                            ELSIF (instHome.Error = TRUE OR instTimerTON.Q) THEN
                                // Errorhandling
                                statStatus                    := ERR_MC_HOME;
                                statErrorAutoCleared          := TRUE;
                                diagnostics                   := statDiagnostics;
                                diagnostics.subfunctionStatus := instHome.ErrorId;
                                statFBState                   := AXIS_STOP_ON_ERROR_SELECTION;
                                statBasicMotionState          := NO_SELECTION;

                            ELSE
                                ; // Command selected

                            END_IF;

                            statExeOfBasicMotion   := 16#0;
                            statExeOfBasicMotion.0 := instHome.Busy;
                            statExeOfBasicMotion.1 := instHome.Done;
                            statExeOfBasicMotion.2 := instHome.CommandAborted;
                            statExeOfBasicMotion.3 := instHome.Error;
                        {END_REGION}
                        HOMING_ON_FIXED_STOP:
                            // This case is additional feature (MC_MOVEVELOCITY and MC_HOME internal used)
                            {REGION "REFERENCE_TO_FIXED_STOP"}
                            CASE statExeOfBasicMotion OF
                                CMD_BUSY:
                                    // Firstcycle of command
                                    IF (statFirstCycleBasicMotion = TRUE) THEN
                                        // Check if homing on fixed stop is allowed  
                                        (*IF ( axis.Modulo.Enable = TRUE) THEN*)
                                        IF (tempFalse = TRUE) THEN
                                            // Modulo enabled - Errorhandling
                                            statStatus                    := ERR_MODULO_NOT_ALLOWED;
                                            statErrorAutoCleared          := TRUE;
                                            diagnostics.subfunctionStatus := 0;
                                            diagnostics.basicMotionState  := statBasicMotionState;
                                            // Set next state
                                            statFBState           := AXIS_STOP_ON_ERROR_SELECTION;
                                            statBasicMotionState  := NO_SELECTION;
                                            statActiveHomingState := STANDARD_HOMING;
                                            statHomingSubState    := HOMING_IDLE;

                                        ELSIF (configuration.homing.extendedModeTorqueLimit = 0) // Torqueliming 0 in configuration 
                                            THEN
                                            // Errorhandling -  Torquevalue 0 configured
                                            statStatus                    := ERR_INVALID_TORQUE_LIMIT;
                                            statErrorAutoCleared          := TRUE;
                                            diagnostics.subfunctionStatus := 0;
                                            diagnostics.basicMotionState  := statBasicMotionState;
                                            // Set next state
                                            statFBState           := AXIS_STOP_ON_ERROR_SELECTION;
                                            statBasicMotionState  := NO_SELECTION;
                                            statActiveHomingState := STANDARD_HOMING;
                                            statHomingSubState    := HOMING_IDLE;

                                            (*ELSIF ( axis.Homing.ReferencingVelocity = 0)*)
                                        ELSIF (configuration.homing.offsetPositionVelocity = 0)
                                            THEN
                                            // Errorhandling -  Velocity 0 configured
                                            statStatus                    := ERR_INVALID_VELOCITY;
                                            statErrorAutoCleared          := TRUE;
                                            diagnostics.subfunctionStatus := 0;
                                            diagnostics.basicMotionState  := statBasicMotionState;
                                            // Set next state
                                            statFBState           := AXIS_STOP_ON_ERROR_SELECTION;
                                            statBasicMotionState  := NO_SELECTION;
                                            statActiveHomingState := STANDARD_HOMING;
                                            statHomingSubState    := HOMING_IDLE;

                                        ELSE
                                            // Store dynamic values
                                            (*statHomingPosition :=  configuration.homing.position;
	                             statVelocity :=  axis.Homing.ReferencingVelocity;
	                             statAcceleration :=  axis.DynamicDefaults.Acceleration;
	                             statDeceleration :=  axis.DynamicDefaults.Deceleration;
	                             statJerk :=  axis.DynamicDefaults.Jerk;
	                             statTorqueLimit :=  configuration.homing.extendedModeTorqueLimit;*)
                                            statHomingPosition := configuration.homing.position;
                                            statVelocity       := configuration.homing.offsetPositionVelocity;
                                            statAcceleration   := configuration.homing.offsetPositionAcceleration;
                                            statDeceleration   := configuration.homing.offsetPositonDeceleration;
                                            statJerk           := configuration.homing.offsetPositionJerk;
                                            statTorqueLimit    := configuration.homing.extendedModeTorqueLimit;

                                            // Detecting operating sensor
                                            (*
								FOR  tempIndex := 1 TO 4 DO
	                              IF  axis.StatusSensor[ tempIndex].Control = TRUE
	                              THEN
	                                EXIT;
	                              END_IF;
	                            END_FOR;
	                            *)
                                            (*IF ( axis.Sensor[ tempIndex].ActiveHoming.Direction = 0) // Positve direction configured
	                            THEN*)
                                            // Positive direction
                                            statDirection := FORWARD_DIR;
                                            (* ELSE
	                              // Negative direction
	                               statDirection :=  BACKWARD_DIR;
	                            END_IF;
	                            *)
                                            (*statTorqueLimitingState :=  FIXED_STOP_DETECTION_ACTIVE;*)
                                            // Reset MC_Commands
                                            instHome(Axis := axis,
                                                     bCalibrationCam := homingSensor,
                                                     Execute := FALSE);

                                            instMoveVelocity(Axis := axis,
                                                             Execute := FALSE);

                                            instMoveAbsolute(Axis := axis,
                                                             Execute := FALSE);

                                            // Reset TON
                                            instTimerTON(IN := FALSE,
                                                         PT := configuration.homing.homeExecutionTimeLimit);

                                            // Determine the encoder type
                                            (* tempIndex := 1;
	                             tempIndex := UDINT_TO_INT( axis.OperativeSensor);
	                            IF ( axis.Sensor[ tempIndex].Type =  INCREMENTAL_ENCODER) THEN
	                               statHomingMode :=  DIRECT_HOMING; // Direct homing (absolute)
	                            ELSE
	                               statHomingMode :=  ABSOLUTE_ENCODER_ADJUSTMENT;
	                            END_IF;
								*)
                                            // Use always direct homing
                                            // statHomingMode :=  DIRECT_HOMING; // Direct homing (absolute)
                                            // Set next state
                                            (*statHomingSubState :=  HOMING_FIXED_STOP_DETECTION;*)
                                            statHomingSubState := HOMING_PROCESS;
                                        END_IF;
                                    END_IF;

                                    // Call OF subStateMachine
                                    REPEAT
                                        CASE statHomingSubState OF
                                            HOMING_IDLE:
                                                tempStateChangeActive := FALSE;
                                                ; // Do nothing, inserted no exectution of homing if error occurred in first cycle

                                            HOMING_FIXED_STOP_DETECTION:
                                                tempStateChangeActive := FALSE;

                                                // Start axis to detect fixed stop
                                                instMoveVelocity(Axis := axis,
                                                                 Execute := TRUE,
                                                                 Velocity := statVelocity,
                                                                 Acceleration := statAcceleration,
                                                                 Deceleration := statDeceleration,
                                                                 Jerk := statJerk,
                                                (*PositionControlled := TRUE,*)
                                                (*Direction :=  statDirection*) );

                                                // Read Statusword only when not already read out
                                                IF (tempStatusWord = 16#0)
                                                    THEN
                                                    (*tempStatusWord :=  axis.StatusWord;*)
                                                    tempStatusWord := axis.NcToPlc.StateDWord;
                                                END_IF;

                                                // Evaluate MC_Command
                                                IF (tempStatusWord.30 = TRUE) THEN // inClamping = TRUE
                                                    // Fixed stop detected --> start homing process
                                                    statHomingSubState    := HOMING_PROCESS;
                                                    tempStateChangeActive := TRUE;

                                                ELSIF (instMoveVelocity.Error = TRUE) THEN
                                                    // Errorhandling
                                                    statStatus                    := ERR_MC_MOVEVELOCITY;
                                                    statErrorAutoCleared          := TRUE;
                                                    diagnostics                   := statDiagnostics;
                                                    diagnostics.subfunctionStatus := instMoveVelocity.ErrorId;
                                                    // Set next state
                                                    statFBState           := AXIS_STOP_ON_ERROR_SELECTION;
                                                    statBasicMotionState  := NO_SELECTION;
                                                    statActiveHomingState := STANDARD_HOMING;
                                                    statExeOfBasicMotion  := CMD_ERROR;
                                                    statHomingSubState    := HOMING_IDLE;

                                                ELSIF (instMoveVelocity.CommandAborted = TRUE) THEN
                                                    // Set next state
                                                    statExeOfBasicMotion := CMD_ABORTED;
                                                    statHomingSubState   := HOMING_IDLE;

                                                ELSE
                                                    ; // Wait for detecting fixed stop
                                                END_IF;

                                            HOMING_PROCESS:
                                                tempStateChangeActive := FALSE;
                                                // Execute MC_HOME
                                                instHome(Axis := axis,
                                                         bCalibrationCam := homingSensor,
                                                         Execute := TRUE,
                                                         Position := statHomingPosition,
                                                (*Mode :=  statHomingMode*) );

                                                //Call TON
                                                instTimerTON(IN := TRUE,
                                                             PT := configuration.homing.homeExecutionTimeLimit);

                                                // Evaluate MC_Command
                                                IF (instHome.Done = TRUE) THEN
                                                    // MC_HOME finished - Set next state
                                                    statHomingSubState    := HOMING_POSITION;
                                                    tempStateChangeActive := TRUE;
                                                    instTimerTON.IN       := FALSE;

                                                ELSIF (instHome.Error = TRUE OR instTimerTON.Q) THEN
                                                    // Errorhandling
                                                    statStatus                    := ERR_MC_HOME;
                                                    statErrorAutoCleared          := TRUE;
                                                    diagnostics                   := statDiagnostics;
                                                    diagnostics.subfunctionStatus := instHome.ErrorId;
                                                    // Set next state
                                                    statFBState          := AXIS_STOP_ON_ERROR_SELECTION;
                                                    statExeOfBasicMotion := CMD_ERROR;
                                                    statHomingSubState   := HOMING_IDLE;

                                                ELSIF (instHome.CommandAborted = TRUE) THEN
                                                    // Set next state
                                                    statExeOfBasicMotion := CMD_ABORTED;
                                                    statHomingSubState   := HOMING_IDLE;
                                                ELSE
                                                    ; // Wait for finish homing process
                                                END_IF;

                                            HOMING_POSITION:
                                                tempStateChangeActive := FALSE;

                                                statHomingPosition := configuration.homing.offsetPosition;
                                                statVelocity       := configuration.homing.offsetPositionVelocity;
                                                statAcceleration   := configuration.homing.offsetPositionAcceleration;
                                                statDeceleration   := configuration.homing.offsetPositonDeceleration;
                                                statJerk           := configuration.homing.offsetPositionJerk;

                                                // Execute moving to homeposition
                                                instMoveAbsolute(Axis := axis,
                                                                 Execute := TRUE,
                                                                 (*Position :=  statHomingPosition,*)
                                                                 Position := configuration.homing.offsetPosition,
                                                                 Velocity := ABS(statVelocity),
                                                                 Acceleration := statAcceleration,
                                                                 Deceleration := statDeceleration,
                                                                 Jerk := statJerk,
                                                (*Direction :=  SHORTEST_WAY_DIR*) );

                                                // Evaluate MC_Command
                                                IF (instMoveAbsolute.Done = TRUE) THEN
                                                    // Homeposition reached - Set next state
                                                    statExeOfBasicMotion := CMD_DONE;
                                                    statHomingSubState   := HOMING_IDLE;

                                                ELSIF (instMoveAbsolute.Error = TRUE) THEN
                                                    // Errorhandling
                                                    statStatus                    := ERR_MC_MOVEABSOLUTE;
                                                    statErrorAutoCleared          := TRUE;
                                                    diagnostics                   := statDiagnostics;
                                                    diagnostics.subfunctionStatus := instMoveAbsolute.ErrorId;
                                                    // Set next state
                                                    statFBState           := AXIS_STOP_ON_ERROR_SELECTION;
                                                    statBasicMotionState  := CMD_BUSY;
                                                    statActiveHomingState := STANDARD_HOMING;
                                                    statExeOfBasicMotion  := CMD_ERROR;
                                                    statHomingSubState    := HOMING_IDLE;

                                                ELSIF (instMoveAbsolute.CommandAborted = TRUE) THEN
                                                    // Set next state
                                                    statExeOfBasicMotion := CMD_ABORTED;
                                                    statHomingSubState   := HOMING_IDLE;

                                                ELSE
                                                    ; // Wait for reaching homeposition
                                                END_IF;

                                        ELSE
                                            // Errorhandling 
                                            statStatus                    := ERR_UNDEFINED_EXTENDED_HOMING_SUBSTATE;
                                            statErrorUserCleared          := TRUE;
                                            diagnostics                   := statDiagnostics;
                                            diagnostics.subfunctionStatus := 0;
                                            // Set errorstate
                                            statFBState           := FB_ERROR;
                                            tempStateChangeActive := FALSE;
                                        END_CASE;

                                    UNTIL (tempStateChangeActive = FALSE) // Repeat execution if a state is changing
                                    END_REPEAT;

                                CMD_DONE,
                                    CMD_ABORTED,
                                    CMD_ERROR:
                                    // Return to NO_SELECTION if command finished
                                    IF (statBasicCommand.10 = FALSE) // homing = FALSE
                                        THEN
                                        // Return to NO_HOMING_ACTIVE if command finished
                                        statBasicMotionState  := NO_SELECTION;
                                        statActiveHomingState := STANDARD_HOMING;
                                        statExeOfBasicMotion  := CMD_BUSY;
                                        statHomingSubState    := HOMING_IDLE;
                                    ELSE
                                        ; // Wait for falling edge at homing command
                                    END_IF;

                            ELSE
                                // Errorhandling
                                statStatus                    := ERR_UNDEFINED_EXTENDED_HOMING_STATE;
                                statErrorUserCleared          := TRUE;
                                diagnostics                   := statDiagnostics;
                                diagnostics.subfunctionStatus := 0;
                                // Set errorstate
                                statFBState := FB_ERROR;
                            END_CASE;
                    {END_REGION}

                    ELSE
                        // Errorhandling
                        statStatus                    := ERR_INVALID_HOMING_EXTENDED_MODE;
                        statErrorAutoCleared          := TRUE;
                        diagnostics                   := statDiagnostics;
                        diagnostics.subfunctionStatus := 0;
                        // Set next state
                        statFBState           := AXIS_STOP_ON_ERROR_SELECTION;
                        statBasicMotionState  := NO_SELECTION;
                        statActiveHomingState := STANDARD_HOMING;
                        statBasicMotionState  := NO_SELECTION;
                    END_CASE;
                {END_REGION}

                GEAR_IN_RELATIVE_SELECTED:
                    // Additional features (applicative): Change setpoint on the fly (gear ratio)
                    {REGION "GEAR_IN_RELATIVE_SELECTED"}
                    // Firstcycle of command
                    IF (statFirstCycleBasicMotion = TRUE) THEN
                        // Reset GEAR_IN command 
                        instGearIn(Master := master,
                                   Slave := axis,
                                   Execute := FALSE);

                        (*statRatioNumerator :=  configuration.gearInRelative.ratioNumerator;*)
                        statRatioNumerator      := configuration.gearInRelative.ratioDenominator;
                        statRatioDenominator    := configuration.gearInRelative.ratioDenominator;
                        statAcceleration        := configuration.gearInRelative.acceleration;
                        statDeceleration        := configuration.gearInRelative.deceleration;
                        statJerk                := configuration.gearInRelative.jerk;
                        statRatioChangeOnTheFly := configuration.gearInRelative.ratioChangeOnTheFly;

                    ELSIF ((statRatioChangeOnTheFly = TRUE) // Flying change of ratio numerator
                    (*AND (( configuration.gearInRelative.ratioNumerator <>  statRatioNumerator)*)
                        AND
                        ((configuration.gearInRelative.ratioDenominator <> statRatioNumerator) OR
                        (configuration.gearInRelative.ratioDenominator <> statRatioDenominator))) AND
                        (instGearIn.CommandAborted = FALSE)
                        THEN
                        instGearIn(Master := master,
                                   Slave := axis,
                                   Execute := FALSE);

                        statRatioNumerator   := configuration.gearInRelative.ratioDenominator; // Apply the new gear ratio numerator
                        statRatioDenominator := configuration.gearInRelative.ratioDenominator; // Apply the new gear ratio denominator
                    END_IF;

                    // Call MC_Command
                    instGearIn(Master := master,
                               Slave := axis,
                               Execute := statBasicCommand.7 OR statFirstCycleBasicMotion, // Input: gearInRelative
                               RatioNumerator := statRatioNumerator,
                               RatioDenominator := DINT_TO_UINT(statRatioDenominator),
                               Acceleration := statAcceleration,
                               Deceleration := statDeceleration,
                               Jerk := statJerk);

                    // Evaluate MC_Command
                    IF (instGearIn.Busy = FALSE) AND
                        (instGearIn.Error = FALSE) AND
                        (instGearIn.CommandAborted = FALSE) AND
                        (instGearIn.InGear = FALSE)
                        THEN
                        // Return to NO_SELECTION if command finished
                        statBasicMotionState := NO_SELECTION;

                    ELSIF (instGearIn.Error = TRUE) THEN
                        // Errorhandling
                        statStatus                    := ERR_MC_GEARIN;
                        statErrorAutoCleared          := TRUE;
                        diagnostics                   := statDiagnostics;
                        diagnostics.subfunctionStatus := instGearIn.ErrorId;
                        statRatioChangeOnTheFly       := FALSE;
                        // Set next state
                        statFBState          := AXIS_STOP_ON_ERROR_SELECTION;
                        statBasicMotionState := NO_SELECTION;

                    ELSE
                        ; // Command selected
                    END_IF;

                    // Read Statusword only when not already read out
                    // IF ( tempStatusWord = 16#0)
                    // THEN
                    //    tempStatusWord :=  axis.StatusWord;
                    // END_IF;

                    // Write MC_Command outputs to internal variable
                    statExeOfBasicMotion   := 16#0;
                    statExeOfBasicMotion.0 := instGearIn.Busy;
                    statExeOfBasicMotion.2 := instGearIn.CommandAborted;
                    statExeOfBasicMotion.3 := instGearIn.Error;
                    // statExeOfBasicMotion.6 :=  tempStatusWord.21 AND NOT  instGearIn.InGear; // write Synchronizing only when bit of instance of MC_GearIn.InGear = FALSE
                    statExeOfBasicMotion.7 := instGearIn.InGear;
                {END_REGION}

                GEAR_IN_ABSOLUTE_SELECTED:
                    // Additional features (applicative): Change setpoint on the fly (gear ratio)
                    {REGION "GEAR_IN_SELECTED"}
                    // Firstcycle of command
                    IF (statFirstCycleBasicMotion = TRUE) THEN
                        // Reset GEAR_IN_POS command 
                        instGearInPos(Master := master,
                                      Slave := axis,
                        (*Execute := FALSE*) );

                        statRatioNumerator       := configuration.gearInAbsolute.ratioNumerator;
                        statRatioDenominator     := configuration.gearInAbsolute.ratioDenominator;
                        statMasterSyncPosition   := configuration.gearInAbsolute.masterSyncPosition;
                        statSlaveSyncPosition    := configuration.gearInAbsolute.slaveSyncPosition;
                        statSyncProfileReference := configuration.gearInAbsolute.syncProfileReference;
                        statMasterStartDistance  := configuration.gearInAbsolute.masterStartDistance;
                        statVelocity             := configuration.gearInAbsolute.velocity;
                        statAcceleration         := configuration.gearInAbsolute.acceleration;
                        statDeceleration         := configuration.gearInAbsolute.deceleration;
                        statJerk                 := configuration.gearInAbsolute.jerk;
                        statSyncDirection        := configuration.gearInAbsolute.syncDirection;
                        statRatioChangeOnTheFly  := configuration.gearInAbsolute.ratioChangeOnTheFly;

                    ELSIF (((statRatioChangeOnTheFly = TRUE) AND (configuration.gearInAbsolute.ratioNumerator <> statRatioNumerator)) OR
                        ((statRatioChangeOnTheFly = TRUE) AND (configuration.gearInAbsolute.ratioDenominator <> statRatioDenominator))) AND
                        (instGearInPos.CommandAborted = FALSE)
                        THEN
                        instGearInPos(Master := master,
                                      Slave := axis,
                        (*Execute := FALSE*) );

                        statRatioNumerator   := configuration.gearInAbsolute.ratioNumerator;   // Apply the new gear ratio numerator
                        statRatioDenominator := configuration.gearInAbsolute.ratioDenominator; // Apply the new gear ratio denominator
                    END_IF;

                    // Call MC_Command
                    instGearInPos(Master := master,
                                  Slave := axis,
                                  Enable := statBasicCommand.8 OR statFirstCycleBasicMotion, // Input: gearInAbsolute
                                  GearRatio := statRatioNumerator,
                                  (*RatioDenominator :=  statRatioDenominator,*)
                                  (*MasterSyncPosition :=  statMasterSyncPosition,*)
                                  (*SlaveSyncPosition :=  statSlaveSyncPosition,*)
                                  (*SyncProfileReference :=  statSyncProfileReference,*)
                                  (*MasterStartDistance :=  statMasterStartDistance,*)
                                  (*Velocity :=  statVelocity,*)
                                  (*Acceleration :=  statAcceleration,*)
                                  (*Deceleration :=  statDeceleration,*)
                                  Jerk := statJerk,
                    (*SyncDirection :=  statSyncDirection*) );

                    // Evaluate MC_Command
                    IF (instGearInPos.Busy = FALSE) AND
                        (instGearInPos.Error = FALSE) AND
                        (instGearInPos.CommandAborted = FALSE) AND
                    (*( instGearInPos.StartSync = FALSE) AND*)
                        (instGearInPos.InGear = FALSE)
                        THEN
                        // Return to NO_SELECTION if command finished
                        statBasicMotionState := NO_SELECTION;

                    ELSIF (instGearInPos.Error = TRUE) THEN
                        // Errorhandling
                        statStatus                    := ERR_MC_GEARINPOS;
                        statErrorAutoCleared          := TRUE;
                        diagnostics                   := statDiagnostics;
                        diagnostics.subfunctionStatus := instGearInPos.ErrorId;
                        statRatioChangeOnTheFly       := FALSE;
                        // Set next state
                        statFBState          := AXIS_STOP_ON_ERROR_SELECTION;
                        statBasicMotionState := NO_SELECTION;

                    ELSE
                        ; // Command selected
                    END_IF;

                    // Write MC_Command outputs to internal variable
                    statExeOfBasicMotion   := 16#0;
                    statExeOfBasicMotion.0 := instGearInPos.Busy;
                    statExeOfBasicMotion.2 := instGearInPos.CommandAborted;
                    statExeOfBasicMotion.3 := instGearInPos.Error;
                    (*statExeOfBasicMotion.6 :=  instGearInPos.StartSync;*)
                    (*statExeOfBasicMotion.6 :=  instGearInPos.StartSync;*)
                    statExeOfBasicMotion.7 := instGearInPos.InGear;
                {END_REGION}

                CAM_IN_SELECTED:
                    // Additional feature (applicative): Check DB of Cam 
                    {REGION "CAM_IN_SELECTED"}
                    // Firstcycle of command
                    IF (statFirstCycleBasicMotion = TRUE) THEN
                        (*IF TypeOfDB( cam) = TO_Cam*)
                        IF tempFalse = FALSE
                            THEN
                            (*statCam :=  cam;*)
                            // Reset CAM_IN command 
                            instCamIn(Master := master,
                                      Slave := axis,
                                      (*Cam :=  statCam,*)
                                      Execute := FALSE);

                            statApplicativeBasicMotionError := FALSE;
                            statApplicationMode             := configuration.camIn.applicationMode;
                        ELSE
                            // Errorhandling - Invalid cam
                            statStatus                      := ERR_INVALID_CAM;
                            statErrorAutoCleared            := TRUE;
                            diagnostics.subfunctionStatus   := 0;
                            diagnostics                     := statDiagnostics;
                            statApplicativeBasicMotionError := TRUE;
                            // Set next state
                            statFBState          := AXIS_STOP_ON_ERROR_SELECTION;
                            statBasicMotionState := NO_SELECTION;
                        END_IF;
                    END_IF;

                    IF (statApplicativeBasicMotionError = FALSE) THEN

                        // Write MC Parameters
                        instCamIn.CamTableID                 := configuration.camIn.tableID;
                        instCamIn.StartMode                  := configuration.camIn.startMode;
                        instCamIn.MasterOffset               := configuration.camIn.masterOffset;
                        instCamIn.SlaveOffset                := configuration.camIn.slaveOffset;
                        instCamIn.MasterScaling              := configuration.camIn.masterScaling;
                        instCamIn.SlaveScaling               := configuration.camIn.slaveScaling;
						instCamIn.StartMode     			 := configuration.camIn.startMode;
                        instCamIn.Options.ActivationMode     := configuration.camIn.ActivationMode;
                        instCamIn.Options.ActivationPosition := configuration.camIn.ActivationPosition;

                        // Call MC_Command
                        instCamIn(Master := master,
                                  Slave := axis,
                                  Execute := statBasicCommand.9 OR statFirstCycleBasicMotion);

                        // Evaluate MC_Command
                        IF ((instCamIn.Busy = FALSE) AND
                            (instCamIn.Error = FALSE) AND
                            (instCamIn.CommandAborted = FALSE) AND
                            (instCamIn.InSync = FALSE) AND
                        (*( instCamIn.StartSync = FALSE) AND*)
                            (statBasicCommand.9 = FALSE)
                            ) AND // V1.0.2 Wait for one cycle EndOfProfile (--> Done) before function is finished at applicationMode ONCE
                            ((statApplicationMode <> APPLICATION_MODE_ONCE) OR
                            ((statApplicationMode = APPLICATION_MODE_ONCE) (*AND ( instCamIn.EndOfProfile = FALSE)*) ))
                            THEN
                            // Return to NO_SELECTION if command finished
                            statBasicMotionState := NO_SELECTION;

                        ELSIF (instCamIn.Error = TRUE) THEN
                            // Errorhandling
                            statStatus                    := ERR_MC_CAMIN;
                            statErrorAutoCleared          := TRUE;
                            diagnostics.subfunctionStatus := instCamIn.ErrorId;
                            diagnostics.basicMotionState  := statBasicMotionState;
                            statFBState                   := AXIS_STOP_ON_ERROR_SELECTION;
                            statBasicMotionState          := NO_SELECTION;

                        ELSE
                            ; // Command selected
                        END_IF;

                        // Write MC_Command outputs to internal variable
                        statExeOfBasicMotion   := 16#0;
                        statExeOfBasicMotion.0 := instCamIn.Busy;
                        IF (statApplicationMode = APPLICATION_MODE_ONCE)
                            THEN
                            ; (*statExeOfBasicMotion.1 :=  instCamIn.EndOfProfile;*)
                        END_IF;

                        statExeOfBasicMotion.2 := instCamIn.CommandAborted;
                        statExeOfBasicMotion.3 := instCamIn.Error;
                        statExeOfBasicMotion.6 := NOT instCamIn.Active;
                        statExeOfBasicMotion.7 := instCamIn.InSync;

                    ELSE
                        ; // InValid cam
                    END_IF;
            {END_REGION}

            ELSE
                // Errorhandling
                statStatus                    := ERR_UNDEFINED_BASIC_MOTION_STATE;
                statErrorUserCleared          := TRUE;
                diagnostics                   := statDiagnostics;
                diagnostics.subfunctionStatus := 0;
                // Set errorstate
                statFBState := FB_ERROR;
            END_CASE;

        RESET_GEARING:
            // Abort waiting absolute gearing / camIn job if new basic motion job is selected (configuration.generalSettings.abortWaitingSyncCmd = TRUE)
            instGearIn(Master := master,
                       Slave := axis,
                       Execute := TRUE,
                       RatioNumerator := 1,
                       RatioDenominator := 1); // Lowest possible gear ratio

            IF (instGearIn.InGear = TRUE) OR (instGearIn.CommandAborted = TRUE)
                THEN                                            // Relative gearing command has aborted waiting absolute gearing job
                statMainSelectionState    := CALL_BASIC_MOTION; // Execute new basic motion command
                tempStateChangeActive     := TRUE;
                statFirstCycleBasicMotion := TRUE;

            ELSIF (instGearIn.Error = TRUE)
                THEN
                statStatus                    := ERR_MC_GEARIN;
                diagnostics.subfunctionStatus := instGearIn.ErrorId;
                // Errorhandling
                statErrorAutoCleared := TRUE;
                diagnostics          := statDiagnostics;
                // Set next state
                statFBState            := AXIS_STOP_ON_ERROR_SELECTION;
                statMainSelectionState := CALL_BASIC_MOTION;
                statBasicMotionState   := NO_SELECTION;

            ELSE
                ; // Command running
            END_IF;

            // Write MC_Command outputs to internal variable
            statExeOfBasicMotion   := 16#0;
            statExeOfBasicMotion.0 := instGearIn.Busy;
    ELSE
        // Errorhandling
        statStatus                    := ERR_UNDEFINED_MAIN_SELECTION_STATE;
        statErrorUserCleared          := TRUE;
        diagnostics                   := statDiagnostics;
        diagnostics.subfunctionStatus := 0;
        // Set errorstate
        statFBState := FB_ERROR;
    END_CASE;

UNTIL (tempStateChangeActive = FALSE)
END_REPEAT;

{END_REGION}

//----------------------------------------------------------------------------------------------
// Execution of homing functionality 
//----------------------------------------------------------------------------------------------
{REGION "EXECUTION_OF_PASSIVE_HOMING"}
// Statemachine for homing functionality
CASE statPassiveHomingState OF
    // Selection of extended homing mode  
    NO_HOMING_ACTIVE:
        ; // Do nothing

    STANDARD_HOMING:
        // No additional features
        {REGION "STANDARD_HOMING"}
        // Firstcycle of command
        IF (statFirstCycleHoming = TRUE) THEN
            // Reset MC_HOME command
            instHome(Axis := axis,
                     bCalibrationCam := homingSensor,
                     Execute := FALSE);

            IF (statBasicMotionState = ACTIVE_HOMING_SELECTED) THEN
                statBasicMotionState := NO_SELECTION;
            END_IF;
        END_IF;

        // Call MC_Command
        instHome(Axis := axis,
                 bCalibrationCam := homingSensor,
                 Execute := statExtendedCommand.2, // Input: homing
                 Position := configuration.homing.position,
        (*Mode :=  configuration.homing.mode*) );

        // Evaluate MC_Command
        IF (instHome.Busy = FALSE) AND
            (instHome.Done = FALSE) AND
            (instHome.CommandAborted = FALSE) AND
            (instHome.Error = FALSE)
            THEN
            // Return to NO_SELECTION if command finished
            statPassiveHomingState := NO_HOMING_ACTIVE;

        ELSIF (instHome.Error = TRUE) THEN
            // Errorhandling
            statStatus                    := ERR_MC_HOME;
            statErrorAutoCleared          := TRUE;
            diagnostics                   := statDiagnostics;
            diagnostics.subfunctionStatus := instHome.ErrorId;
            statPassiveHomingState        := NO_HOMING_ACTIVE;
            // Set next state
            statFBState := AXIS_STOP_ON_ERROR_SELECTION;
        ELSE
            ; // Command selected

        END_IF;

        statExeOfHoming   := 16#0;
        statExeOfHoming.0 := instHome.Busy;
        statExeOfHoming.1 := instHome.Done;
        statExeOfHoming.2 := instHome.CommandAborted;
        statExeOfHoming.3 := instHome.Error;
{END_REGION}

ELSE
    // Errorhandling
    statStatus                              := ERR_INVALID_HOMING_EXTENDED_MODE;
    statErrorAutoCleared                    := TRUE;
    diagnostics                             := statDiagnostics;
    diagnostics.subfunctionStatus           := 0;
    statDiagnostics.basicMotionState        := statBasicMotionState;
    statDiagnostics.superimposedMotionState := statSupImpMotionState;
    // Set next state
    statFBState            := AXIS_STOP_ON_ERROR_SELECTION;
    statBasicMotionState   := NO_SELECTION;
    statPassiveHomingState := NO_HOMING_ACTIVE;
END_CASE;

{END_REGION}

//----------------------------------------------------------------------------------------------
// Execution of functionalities of superimposed coordinate system
//----------------------------------------------------------------------------------------------
{REGION "EXECUTION_OF_SUPERIMPOSED_COMMANDS"}
// Statemachine for superimposed motion commands
// Write diagnostics
statDiagnostics.basicMotionState        := statBasicMotionState;
statDiagnostics.superimposedMotionState := statSupImpMotionState;

CASE statSupImpMotionState OF
    NO_SELECTION:
        ; // Do nothing

    POS_SUPERIMPOSED_SELECTED:
        // Additional features (applicative) : Specified direction
        {REGION "POS_SUPERIMPOSED_SELECTED;"}
        // Firstcycle of command
        IF (statFirstCycleSupImpMotion = TRUE) THEN
            // Configurate the direction of rotation
            IF ((configuration.posSuperimposed.direction = 0) AND (configuration.posSuperimposed.distance >= 0.0)) // Sign of distance is evaluated
                OR
                (configuration.posSuperimposed.direction = FORWARD_DIR) // Positive direction
                THEN
                statSupImpMotionPosition := ABS(configuration.posSuperimposed.distance);
                // Reset MC_MOVESUPERIMPOSED command
                instMoveSuperimposed(Axis := axis,
                                     Execute := FALSE);

                statApplicativeSupImpMotionError := FALSE;
            ELSIF ((configuration.posSuperimposed.direction = 0) AND (configuration.posSuperimposed.distance < 0.0)) // Sign of distance is evaluated
                OR
                (configuration.posSuperimposed.direction = BACKWARD_DIR) // Negative direction 
                THEN
                statSupImpMotionPosition := -ABS(configuration.posSuperimposed.distance);
                // Reset MC_MOVESUPERIMPOSED command
                instMoveSuperimposed(Axis := axis,
                                     Execute := FALSE);

                statApplicativeSupImpMotionError := FALSE;

            ELSE
                // Errorhandling - Invalid direction
                statStatus                       := ERR_INVALID_POS_SUPERIMPOSED_DIR;
                statErrorAutoCleared             := TRUE;
                diagnostics                      := statDiagnostics;
                diagnostics.subfunctionStatus    := 0;
                statApplicativeSupImpMotionError := TRUE;
                // Set next state
                statFBState           := AXIS_STOP_ON_ERROR_SELECTION;
                statSupImpMotionState := NO_SELECTION;
            END_IF;
        END_IF;

        IF (statApplicativeSupImpMotionError = FALSE) THEN
            // Call MC_Command
            instMoveSuperimposed(Axis := axis,
                                 Execute := statSupImpCommand.0, // Input: posSuperimposed
                                 Distance := statSupImpMotionPosition,
                                 VelocityDiff := configuration.posSuperimposed.velocityDiff,
                                 Acceleration := configuration.posSuperimposed.acceleration,
                                 Deceleration := configuration.posSuperimposed.deceleration,
                                 Jerk := configuration.posSuperimposed.jerk);

            // Evaluate MC_Command
            IF (instMoveSuperimposed.Busy = FALSE) AND
                (instMoveSuperimposed.Error = FALSE) AND
                (instMoveSuperimposed.Done = FALSE) AND
                (instMoveSuperimposed.CommandAborted = FALSE)
                THEN
                // Return to NO_SELECTION if command finished
                statSupImpMotionState := NO_SELECTION;

            ELSIF (instMoveSuperimposed.Error = TRUE) THEN
                // Errorhandling
                statStatus                    := ERR_MC_MOVESUPERIMPOSED;
                statErrorAutoCleared          := TRUE;
                diagnostics                   := statDiagnostics;
                diagnostics.subfunctionStatus := instMoveSuperimposed.ErrorId;
                // Set next state
                statFBState           := AXIS_STOP_ON_ERROR_SELECTION;
                statSupImpMotionState := NO_SELECTION;

            ELSE
                ; // command selected
            END_IF;

            statExeOfSupImpMotionState   := 16#0;
            statExeOfSupImpMotionState.0 := instMoveSuperimposed.Busy;
            statExeOfSupImpMotionState.1 := instMoveSuperimposed.Done;
            statExeOfSupImpMotionState.2 := instMoveSuperimposed.CommandAborted;
            statExeOfSupImpMotionState.3 := instMoveSuperimposed.Error;
        END_IF;
    {END_REGION}

    PHASING_SELECTED:
        // Additional features (applicative) : Change setpoint on the fly (phaseShift)
        {REGION "PHASING_SELECTED"}
        // Firstcycle of command
        IF (statFirstCycleSupImpMotion = TRUE) THEN
            // Reset MC_PHASING_ABSOLUTE command
            instPhasingAbsolute(Master := master,
                                Slave := axis,
                                Execute := FALSE);

            // Reset MC_PHASING_RELATIVE command
            instPhasingRelative(Master := master,
                                Slave := axis,
                                Execute := FALSE);

            statPhaseShift               := configuration.phasing.phaseShift;
            statVelocity                 := configuration.phasing.velocity;
            statAcceleration             := configuration.phasing.acceleration;
            statDeceleration             := configuration.phasing.deceleration;
            statJerk                     := configuration.phasing.jerk;
            statPhaseAbsolute            := configuration.phasing.phaseAbsolute;
            statChangePhaseShiftOnTheFly := configuration.phasing.phaseShiftChangeOnTheFly;

        ELSIF ((statChangePhaseShiftOnTheFly = TRUE) AND
            (configuration.phasing.phaseShift <> statPhaseShift)) AND
            (statPhaseAbsolute = TRUE) AND
            (instPhasingAbsolute.CommandAborted = FALSE)
            THEN
            // Reset MC_PHASING_ABSOLUTE command - Phaseshift on the fly is only possible at phasing absolut
            instPhasingAbsolute(Master := master,
                                Slave := axis,
                                Execute := FALSE);

            statPhaseShift := configuration.phasing.phaseShift;
        END_IF;

        // Select phasing absolut or relative 
        IF (statPhaseAbsolute = TRUE) THEN
            // Absolute phasing
            // Call MC_Command
            instPhasingAbsolute(Master := master,
                                Slave := axis,
                                Execute := statSupImpCommand.1, // Input: phasing
                                PhaseShift := statPhaseShift,
                                Velocity := statVelocity,
                                Acceleration := statAcceleration,
                                Deceleration := statDeceleration,
                                Jerk := statJerk);

            // Evaluate MC_Command
            IF (instPhasingAbsolute.Busy = FALSE) AND
                (instPhasingAbsolute.Error = FALSE) AND
                (instPhasingAbsolute.Done = FALSE) AND
                (instPhasingAbsolute.CommandAborted = FALSE)
                THEN
                // Return to NO_SELECTION if command finished
                statSupImpMotionState := NO_SELECTION;

            ELSIF (instPhasingAbsolute.Error = TRUE) THEN
                // Errorhandling
                statStatus                    := ERR_MC_PHASINGABSOLUTE;
                statErrorAutoCleared          := TRUE;
                diagnostics                   := statDiagnostics;
                diagnostics.subfunctionStatus := instPhasingAbsolute.ErrorId;
                statChangePhaseShiftOnTheFly  := FALSE;
                // Set next state
                statFBState           := AXIS_STOP_ON_ERROR_SELECTION;
                statSupImpMotionState := NO_SELECTION;

            ELSE
                ; // Command busy
            END_IF;

            statExeOfSupImpMotionState   := 16#0;
            statExeOfSupImpMotionState.0 := instPhasingAbsolute.Busy;
            statExeOfSupImpMotionState.1 := instPhasingAbsolute.Done;
            statExeOfSupImpMotionState.2 := instPhasingAbsolute.CommandAborted;
            statExeOfSupImpMotionState.3 := instPhasingAbsolute.Error;

        ELSE
            // Relative phasing  
            // Call MC_Command
            instPhasingRelative(Master := master,
                                Slave := axis,
                                Execute := statSupImpCommand.1, // Input: phasing
                                PhaseShift := statPhaseShift,
                                Velocity := statVelocity,
                                Acceleration := statAcceleration,
                                Deceleration := statDeceleration,
                                Jerk := statJerk);

            // Evaluate MC_Command
            IF (instPhasingRelative.Busy = FALSE) AND
                (instPhasingRelative.Error = FALSE) AND
                (instPhasingRelative.Done = FALSE) AND
                (instPhasingRelative.CommandAborted = FALSE)
                THEN
                // Return to NO_SELECTION if command finished
                statSupImpMotionState := NO_SELECTION;

            ELSIF (instPhasingRelative.Error = TRUE) THEN
                // Errorhandling
                statStatus                    := ERR_MC_PHASINGRELATIVE;
                statErrorAutoCleared          := TRUE;
                diagnostics                   := statDiagnostics;
                diagnostics.subfunctionStatus := instPhasingRelative.ErrorId;
                statChangePhaseShiftOnTheFly  := FALSE;
                // Set next state
                statFBState           := AXIS_STOP_ON_ERROR_SELECTION;
                statSupImpMotionState := NO_SELECTION;
            ELSE
                ; // Command selected
            END_IF;

            statExeOfSupImpMotionState   := 16#0;
            statExeOfSupImpMotionState.0 := instPhasingRelative.Busy;
            statExeOfSupImpMotionState.1 := instPhasingRelative.Done;
            statExeOfSupImpMotionState.2 := instPhasingRelative.CommandAborted;
            statExeOfSupImpMotionState.3 := instPhasingRelative.Error;
        END_IF;
{END_REGION}

ELSE
    // Errorhandling
    statStatus                    := ERR_UNDEFINED_SUPERIMPOSED_MOTION_STATE;
    statErrorUserCleared          := TRUE;
    diagnostics                   := statDiagnostics;
    diagnostics.subfunctionStatus := 0;
    // Set errorstate
    statFBState := FB_ERROR;
END_CASE;

{END_REGION}

//----------------------------------------------------------------------------------------------
// Execution of torquelimiting functionality
//----------------------------------------------------------------------------------------------
{REGION "EXECUTION_OF_TORQUELIMTING"}
// Statemachine for torquelimiting 
REPEAT
    tempStateChangeActive := FALSE;
    CASE statTorqueLimitingState OF
        NO_TORQUE_LIMITING_ACTIVE:
            ; // Torquelimiting disable
        //  instTorqueLimiting(Axis :=  axis, V01.00.03 Dont Call MC_TORQUELIMITING if disabled
        //                     Enable := FALSE);

        TORQUE_LIMITING_DISABLE:
            // Torquelimiting disable
            instTorqueLimiting(Axis := axis,
                               Enable := FALSE);

            // Check state of torque limting
            IF (instTorqueLimiting.Busy = FALSE)
                THEN
                // set next state
                statTorqueLimitingState := NO_TORQUE_LIMITING_ACTIVE;
            ELSE
                ; // Waiting for MC_Torquelimiting is not busy
            END_IF;

        TORQUE_LIMTING_SELECTED:
            // No extended homing function active
            instTorqueLimiting(Axis := axis,
                               Enable := statExtendedCommand.1,
                               TLimit := configuration.torqueLimiting.TorqueLimit,
                               Mode := configuration.torqueLimiting.mode);

            IF (instTorqueLimiting.Busy = FALSE) THEN
                // Reset state
                statTorqueLimitingState := NO_TORQUE_LIMITING_ACTIVE;
            END_IF;

        (*
	        V1.00.03 Not required anymore
	       AUTOMATIC_MODE_CHANGE:
	        // In this state the torquelimiting function is operating with Mode 1 (Fixed stop detection) until inClamping = FALSE
	         instTorqueLimiting(Axis :=  axis,
	                            Enable := TRUE,
	                            Limit :=  configuration.homing.extendedModeTorqueLimit); // V01.00.03 Always use configured value
	        
	        IF ( configuration.torqueLimiting.mode =  MODE_FIXED_STOP_DETECTION)
	          OR ( instTorqueLimiting.InClamping = FALSE)
	        THEN
	          // Change state
	           statTorqueLimitingState :=  TORQUE_LIMTING_SELECTED;
	           tempStateChangeActive := TRUE;
	        ELSE
	          ; // Wait for InClamping = FALSE
	        END_IF;
	        *)

        FIXED_STOP_DETECTION_ACTIVE:
            // Extended homing function active
            instTorqueLimiting(Axis := axis,
                               Enable := TRUE,
                               TLimit := configuration.homing.extendedModeTorqueLimit, // V01.00.03 Always use configured value
                               Mode := MODE_FIXED_STOP_DETECTION);

            IF ((statHomingSubState = HOMING_IDLE) AND (statBasicMotionState = ACTIVE_HOMING_SELECTED))
                THEN
                // Fixed stop process has finished - Axis is still in clamping
                statTorqueLimitingState := FIXED_STOP_DETECTION_FINISHED;
                tempStateChangeActive   := TRUE;

            ELSIF (statBasicMotionState <> ACTIVE_HOMING_SELECTED)
                THEN
                // Error occurred - change state depending on inClamping
                IF (instTorqueLimiting.InClamping = TRUE)
                    THEN
                    // Axis is in clamping
                    statTorqueLimitingState := FIXED_STOP_DETECTION_ERROR_IN_CLAMPING;
                    tempStateChangeActive   := TRUE;
                ELSE
                    // Axis is in not clamping
                    statTorqueLimitingState := FIXED_STOP_DETECTION_ERROR_NOT_IN_CLAMPING;
                    tempStateChangeActive   := TRUE;
                END_IF;

            ELSE
                ; // Fixed stop detection is running
            END_IF;

        FIXED_STOP_DETECTION_FINISHED:
            // Homing on fixed stop process has finished
            instTorqueLimiting(Axis := axis,
                               Enable := TRUE,
                               TLimit := configuration.homing.extendedModeTorqueLimit, // V01.00.03 Always use configured value
                               Mode := MODE_FIXED_STOP_DETECTION);

            IF (instTorqueLimiting.InClamping = FALSE)
                THEN
                // InClamping = FALSE
                IF (statExtendedCommand.1 = TRUE) // Torquelimiting
                    THEN
                    statTorqueLimitingState := TORQUE_LIMTING_SELECTED;
                ELSE
                    statTorqueLimitingState := TORQUE_LIMITING_DISABLE;
                END_IF;

                tempStateChangeActive := TRUE;
            ELSE
                // InClamping = TRUE
                IF (statExtendedCommand.1 = TRUE) // Torquelimiting
                    AND
                    (configuration.torqueLimiting.mode = MODE_FIXED_STOP_DETECTION)
                    THEN
                    // Change State
                    statTorqueLimitingState := TORQUE_LIMTING_SELECTED;
                    tempStateChangeActive   := TRUE;
                ELSE
                    ; // Wait for inClamping = FALSE
                END_IF;
            END_IF;

        FIXED_STOP_DETECTION_ERROR_IN_CLAMPING:
            // Errorstate, torquelimiting is still active and axis not in clamping
            instTorqueLimiting(Axis := axis,
                               Enable := TRUE,
                               TLimit := configuration.homing.extendedModeTorqueLimit, // V01.00.03 Always use configured value
                               Mode := MODE_FIXED_STOP_DETECTION);

            IF (instTorqueLimiting.InClamping = FALSE)
                THEN
                // InClamping = FALSE -> reset torque limiting state
                statTorqueLimitingState := TORQUE_LIMITING_DISABLE;
                // Torquelimiting disable
                tempStateChangeActive := TRUE;
            END_IF;

        FIXED_STOP_DETECTION_ERROR_NOT_IN_CLAMPING:
            // Errorstate, torquelimiting is still active and axis in clamping
            instTorqueLimiting(Axis := axis,
                               Enable := TRUE,
                               TLimit := configuration.homing.extendedModeTorqueLimit, // V01.00.03 Always use configured value
                               Mode := MODE_FIXED_STOP_DETECTION);

            IF (instTorqueLimiting.InClamping = TRUE)
                THEN
                // InClamping = TRUE -> change state
                statTorqueLimitingState := FIXED_STOP_DETECTION_ERROR_IN_CLAMPING;
                tempStateChangeActive   := TRUE;

            ELSIF (statBasicMotionState <> NO_SELECTION) OR (statSupImpMotionState <> NO_SELECTION) OR (statPassiveHomingState <> NO_HOMING_ACTIVE)
                THEN
                // New valid command is set -> reset error state
                statTorqueLimitingState := TORQUE_LIMITING_DISABLE;
                tempStateChangeActive   := TRUE;

            ELSE
                ; // Waiting for new command or axis is getting in clamping
            END_IF;
    ELSE
        // Errorhandling
        statStatus                          := ERR_UNDEFINED_TORQUE_LIMITING_STATE;
        statErrorUserCleared                := TRUE;
        diagnostics.basicMotionState        := statBasicMotionState;
        diagnostics.superimposedMotionState := statSupImpMotionState;
        diagnostics.subfunctionStatus       := 0;
        // Set errorstate
        statFBState := FB_ERROR;
    END_CASE;
UNTIL (tempStateChangeActive = FALSE)
END_REPEAT;

// Evaluate MC_Command
IF (instTorqueLimiting.Error = TRUE) AND ((statTorqueLimitingErrorOld = FALSE) OR (statStatus = STATUS_SUBSEQUENT_CALL)) THEN
    // Errorhandling
    statStatus                          := ERR_MC_TORQUELIMITING;
    statErrorAutoCleared                := TRUE;
    diagnostics.basicMotionState        := statBasicMotionState;
    diagnostics.superimposedMotionState := statSupImpMotionState;
    diagnostics.subfunctionStatus       := instTorqueLimiting.ErrorId;
    statFBState                         := AXIS_STOP_ON_ERROR_SELECTION;

ELSIF (instTorqueLimiting.Error = FALSE) AND ((statTorqueLimitingErrorOld = TRUE) AND (statStatus = ERR_MC_TORQUELIMITING)) THEN
    statStatus           := STATUS_SUBSEQUENT_CALL;
    statErrorAutoCleared := FALSE;
ELSE
    ;
END_IF;

statTorqueLimitingErrorOld := instTorqueLimiting.Error;
{END_REGION}

//----------------------------------------------------------------------------------------------
// Selection of StopOnError / implementation of fastStop
//----------------------------------------------------------------------------------------------
{REGION "STOP_ON_ERROR"}
// Check for stopping if error occurred during execution of motion commands
IF (statFBState = AXIS_STOP_ON_ERROR_SELECTION)
    THEN
    statBasicMotionState   := NO_SELECTION;
    statSupImpMotionState  := NO_SELECTION;
    statPassiveHomingState := NO_HOMING_ACTIVE;

    IF (configuration.generalSettings.stopOnError = TRUE)
        THEN
        // Read Statusword only when not already read out
        IF (tempStatusWord = 16#0)
            THEN
            tempStatusWord := axis.NcToPlc.StateDWord;
        END_IF;

        // Evaluate error
        IF tempStatusWord.0 THEN
            ; // Axis enabled
            IF (tempStatusWord.1 = TRUE) THEN
                ; // TO Alarm present
                statFBState := AXIS_MOTION;
            ELSE
                // No TO alarm present, set fastStop
                statBasicMotionState      := FAST_STOP_SELECTED;
                statFirstCycleBasicMotion := TRUE;
                statFBState               := AXIS_STOP_ON_ERROR_EXECUTION;
            END_IF;

        ELSE
            ; // Axis disabled
            statFBState := AXIS_MOTION;
        END_IF;

    ELSE
        // Dont StopOnError
        statFBState := AXIS_MOTION;
    END_IF;
END_IF;

// Implementation of fastStop
IF (statBasicMotionState = FAST_STOP_SELECTED) THEN
    // Additional feature: Load emergency stop dynamics (TO) if no valid dynamics are configured for fastStop
    {REGION "FASTSTOP SELECTED"}
    // Firstcycle of command
    IF (statFirstCycleBasicMotion = TRUE) THEN
        // Reset HALT command
        instHalt(Axis := axis,
                 Execute := FALSE);

        statFirstCycleDone := TRUE;
        // Check dynamics for fastStop
        // Load TO emergency Stop dynamics if value <=0 for deceleration is configured
        IF (configuration.fastStop.deceleration <= 0) // V1.0.2 Read TO emergencyStop deceleration only if fastStop.deceleration <= 0
            THEN
            // Invalid fastStop dynamics configured - read emergency stop dynamics from TO
            (*statDeceleration :=  axis.DynamicDefaults.EmergencyDeceleration;*)
            statDeceleration := configuration.fastStop.deceleration;
        ELSE
            // Valid fastStop dynamics configured
            statDeceleration := configuration.fastStop.deceleration;
        END_IF;

        statJerk              := configuration.fastStop.jerk;              // V1.0.2 Use always configuration for jerk value
        statAbortAcceleration := configuration.fastStop.abortAcceleration; // V1.0.2 Use always configuration
    END_IF;

    // Call of MC_Command
    instHalt(Axis := axis,
             Execute := (statBasicCommand.0 OR statFirstCycleBasicMotion),
             Deceleration := statDeceleration,
             (*AbortAcceleration :=  statAbortAcceleration,*)
             Jerk := statJerk);

    // Evaluate MC_Command
    IF (instHalt.Busy = FALSE) AND
        (instHalt.Error = FALSE) AND
        (instHalt.Done = FALSE) AND
        (instHalt.CommandAborted = FALSE)
        THEN
        // Return to NO_SELECTION if command finished
        statFBState          := AXIS_MOTION;
        statBasicMotionState := NO_SELECTION;

    ELSIF (instHalt.Done = TRUE)
        THEN
        IF (statFirstCycleDone = TRUE)
            THEN
            // Command is reset
            IF (instTorqueLimiting.Error = FALSE) // V1.00.03 Dont reset error is pending
                THEN
                // Reset status not if torquelimiting error is pending
                statStatus           := STATUS_SUBSEQUENT_CALL;
                statErrorAutoCleared := FALSE;
            END_IF;

            statFirstCycleDone := FALSE;
        END_IF;

    ELSIF (instHalt.Error = TRUE)
        THEN
        // Errorhandling
        statStatus                          := ERR_MC_HALT;
        statErrorAutoCleared                := TRUE;
        diagnostics                         := statDiagnostics;
        diagnostics.basicMotionState        := statBasicMotionState;
        diagnostics.superimposedMotionState := statSupImpMotionState;
        diagnostics.subfunctionStatus       := instHalt.ErrorId;

    ELSE
        ; // Command selected
    END_IF;

    // Write MC_Command outputs to internal variable
    statExeOfBasicMotion   := 0;
    statExeOfBasicMotion.0 := instHalt.Busy;
    statExeOfBasicMotion.1 := instHalt.Done;
    statExeOfBasicMotion.2 := instHalt.CommandAborted;
    statExeOfBasicMotion.3 := instHalt.Error;
    {END_REGION}
END_IF;

{END_REGION}
//----------------------------------------------------------------------------------------------
// Store values and reset variables
//----------------------------------------------------------------------------------------------
{REGION "STORE_AND_RESET"}
// Reset variables to determine first cycle of a new command
IF (statFirstCycleReset = TRUE) THEN
    statFirstCycleReset := FALSE;
END_IF;

IF (statFirstCycleHoming = TRUE) THEN
    statFirstCycleHoming := FALSE;
END_IF;

statHomingOld := tempHoming;

IF (statFirstCycleBasicMotion = TRUE) THEN
    statFirstCycleBasicMotion := FALSE;
END_IF;

statBasicCommandOld := statBasicCommand;

IF (statFirstCycleSupImpMotion = TRUE) THEN
    statFirstCycleSupImpMotion := FALSE;
END_IF;

statSupImpCommandOld := statSupImpCommand;

// Store last values for edge detection
statEnableOld          := enable;
statEnableAxisOld      := enableAxis;
statExtendedCommandOld := statExtendedCommand;
statPowerErrorOld      := instPower.Error;
{END_REGION}

//----------------------------------------------------------------------------------------------
// Writing outputs
//----------------------------------------------------------------------------------------------
{REGION "WRITING_OF_OUTPUTS"}
// Writing status outputs
resetActive := (statResetState = CMD_BUSY);

IF (statErrorUserCleared = TRUE) THEN
    ; // Reset variables at ErrorUserCleared
    statBasicMotionState       := NO_SELECTION;
    statExeOfBasicMotion       := NO_SELECTION;
    statSupImpMotionState      := NO_SELECTION;
    statExeOfSupImpMotionState := NO_SELECTION;
    statExeOfHoming            := NO_SELECTION;
END_IF;

IF (instPower.Status = TRUE)
    THEN
    // Axis enabled
    axisEnabled := TRUE;

ELSIF (instPower.Error = TRUE) AND (instPower.Status = FALSE)
    THEN
    // Reset status if error occurred
    axisEnabled := FALSE;

ELSIF (instPower.Busy = FALSE)
    THEN
    // Reset if MC_Power is not busy
    axisEnabled := FALSE;
ELSE
    ;
END_IF;

{REGION "WRITING_BASICMOTION_OUTPUTS"}
// Writing Busy, Done and Aborted outputs for basic motion commands
IF (statBasicMotionState > NO_SELECTION) AND (statBasicMotionState < ACTIVE_HOMING_SELECTED)
    THEN
    commandBusy    := statExeOfBasicMotion.0;
    commandDone    := statExeOfBasicMotion.1;
    commandAborted := statExeOfBasicMotion.2;
    inVelocity     := statExeOfBasicMotion.4;
    inSync         := statExeOfBasicMotion.7;
    startSync      := statExeOfBasicMotion.6;
ELSE
    commandBusy    := FALSE;
    commandDone    := FALSE;
    commandAborted := FALSE;
    inVelocity     := FALSE;
    inSync         := FALSE;
    startSync      := FALSE;
END_IF;

// Writing outputs up to LAxisCtrl_SpeedAxis
IF (statTorqueLimitingState = TORQUE_LIMTING_SELECTED)
// OR ( statTorqueLimitingState =  AUTOMATIC_MODE_CHANGE) V1.0.3 TorqueLimtinig = TRUE, only when respective value used 
    THEN
    torqueLimitingSelected := TRUE;
ELSE
    torqueLimitingSelected := FALSE;
END_IF;

inLimitation         := instTorqueLimiting.InLimitation;
fastStopSelected     := statBasicMotionState.0;
stopSelected         := statBasicMotionState.1;
jogSelected          := statBasicMotionState.2 OR statBasicMotionState.3;
moveVelocitySelected := statBasicMotionState.4;
// Writing outputs up to LAxisCtrl_PosAxis
inClamping          := instTorqueLimiting.InClamping;
posRelativeSelected := statBasicMotionState.5;
posAbsoluteSelected := statBasicMotionState.6;
// Writing outputs up to LAxisCtrl_SyncAxisRelGearing
gearInRelativeSelected := statBasicMotionState.7;
// Writing outputs up to LAxisCtrl_SyncAxisCamming
gearInAbsoluteSelected := statBasicMotionState.8;
camInSelected          := statBasicMotionState.9;
//inSimulation           := instSyncMotionSimulation.InSimulation;
{END_REGION}
{REGION "WRITING_HOMING_OUTPUTS"}
// Writing Busy, Done and Aborted outputs for homing
IF (statPassiveHomingState = STANDARD_HOMING)
    THEN
    homingSelected       := TRUE;
    homingCommandBusy    := statExeOfHoming.0;
    homingCommandDone    := statExeOfHoming.1;
    homingCommandAborted := statExeOfHoming.2;
ELSE
    IF (statBasicMotionState = ACTIVE_HOMING_SELECTED)
        THEN
        homingSelected       := TRUE;
        homingCommandBusy    := statExeOfBasicMotion.0;
        homingCommandDone    := statExeOfBasicMotion.1;
        homingCommandAborted := statExeOfBasicMotion.2;
    ELSE
        homingSelected       := FALSE;
        homingCommandBusy    := FALSE;
        homingCommandDone    := FALSE;
        homingCommandAborted := FALSE;
    END_IF;
END_IF;

{END_REGION}
{REGION "WRITING_SUPERIMPOSED_OUTPUTS"}
// Writing outputs for superimposed motion commands
IF (statSupImpMotionState <> NO_SELECTION)
    THEN
    superimposedBusy    := statExeOfSupImpMotionState.0;
    superimposedDone    := statExeOfSupImpMotionState.1;
    superimposedAborted := statExeOfSupImpMotionState.2;
ELSE
    superimposedBusy    := FALSE;
    superimposedDone    := FALSE;
    superimposedAborted := FALSE;
END_IF;

posSuperimposedSelected := statSupImpMotionState.0;
phasingSelected         := statSupImpMotionState.1;
{END_REGION}
{END_REGION}

//----------------------------------------------------------------------------------------------
// Error handling 
//----------------------------------------------------------------------------------------------
{REGION "ERROR_HANDLING"}
IF statErrorUserCleared THEN
    valid              := FALSE;
    busy               := TRUE;
    error              := TRUE;
    status             := statStatus;
    diagnostics.status := statStatus;

ELSIF statErrorAutoCleared THEN
    valid              := FALSE;
    busy               := TRUE;
    error              := TRUE;
    status             := statStatus;
    diagnostics.status := statStatus;

ELSE
    // Process normal output values
    valid  := TRUE;
    error  := FALSE;
    status := statStatus;
END_IF;

{END_REGION}

END_FUNCTION_BLOCK

// ---- Library/FAS/IO-Link/00BW12 - 16 Solenoid Island/_FB_00BW1.TcPOU
FUNCTION_BLOCK _FB_00BW1
VAR_INPUT
	
	solenoid_01 : BOOL;
	solenoid_02 : BOOL;
	solenoid_03 : BOOL;
	solenoid_04 : BOOL;
	solenoid_05 : BOOL;
	solenoid_06 : BOOL;
	solenoid_07 : BOOL;
	solenoid_08 : BOOL;
	solenoid_09 : BOOL;
	solenoid_10 : BOOL;
	solenoid_11 : BOOL;
	solenoid_12 : BOOL;
	solenoid_13 : BOOL;
	solenoid_14 : BOOL;
	solenoid_15 : BOOL;
	solenoid_16 : BOOL;
	solenoid_17 : BOOL;
	solenoid_18 : BOOL;
	solenoid_19 : BOOL;
	solenoid_20 : BOOL;
	solenoid_21 : BOOL;
	solenoid_22 : BOOL;
	solenoid_23 : BOOL;
	solenoid_24 : BOOL;
	solenoid_25 : BOOL;
	solenoid_26 : BOOL;
	solenoid_27 : BOOL;
	solenoid_28 : BOOL;
	solenoid_29 : BOOL;
	solenoid_30 : BOOL;
	solenoid_31 : BOOL;
	solenoid_32 : BOOL;
	
	PlcToHw AT %Q* : _00BW12_PLCTOHW_PDOS;	
		
END_VAR


PlcToHw.outputByte_0.0 := solenoid_01;
PlcToHw.outputByte_0.1 := solenoid_02;
PlcToHw.outputByte_0.2 := solenoid_03;
PlcToHw.outputByte_0.3 := solenoid_04;
PlcToHw.outputByte_0.4 := solenoid_05;
PlcToHw.outputByte_0.5 := solenoid_06;
PlcToHw.outputByte_0.6 := solenoid_07;
PlcToHw.outputByte_0.7 := solenoid_08;

PlcToHw.outputByte_1.0 := solenoid_09;
PlcToHw.outputByte_1.1 := solenoid_10;
PlcToHw.outputByte_1.2 := solenoid_11;
PlcToHw.outputByte_1.3 := solenoid_12;
PlcToHw.outputByte_1.4 := solenoid_13;
PlcToHw.outputByte_1.5 := solenoid_14;
PlcToHw.outputByte_1.6 := solenoid_15;
PlcToHw.outputByte_1.7 := solenoid_16;

PlcToHw.outputByte_2.0 := solenoid_17;
PlcToHw.outputByte_2.1 := solenoid_18;
PlcToHw.outputByte_2.2 := solenoid_19;
PlcToHw.outputByte_2.3 := solenoid_20;
PlcToHw.outputByte_2.4 := solenoid_21;
PlcToHw.outputByte_2.5 := solenoid_22;
PlcToHw.outputByte_2.6 := solenoid_23;
PlcToHw.outputByte_2.7 := solenoid_24;

PlcToHw.outputByte_3.0 := solenoid_25;
PlcToHw.outputByte_3.1 := solenoid_26;
PlcToHw.outputByte_3.2 := solenoid_27;
PlcToHw.outputByte_3.3 := solenoid_28;
PlcToHw.outputByte_3.4 := solenoid_29;
PlcToHw.outputByte_3.5 := solenoid_30;
PlcToHw.outputByte_3.6 := solenoid_31;
PlcToHw.outputByte_3.7 := solenoid_32;

END_FUNCTION_BLOCK

// ---- Library/FAS/IO-Link/0AC001 - Analog Input/_FB_0AC001.TcPOU
FUNCTION_BLOCK _FB_0AC001

VAR_INPUT PERSISTENT

	deviceConfig    : _0AC001_DEV_CONFIG; // Configuration settings for the CT121F device
	
END_VAR
VAR_INPUT 

	  HwToPlc AT %I* : _0AC001_HWTOPLC_PDOS; // Process Data Objects for RWPT01D communication
	
END_VAR
VAR_OUTPUT
	
	analogInput : REAL;
	analogInputRaw : REAL;

END_VAR

_AnalogInputs();

METHOD PRIVATE _AnalogInputs
VAR_INPUT
END_VAR
// Scale sensor distance
analogInput := _Scale(
    X := ((SHL(BYTE_TO_WORD(HwToPlc.inputByte_0),8) OR HwToPlc.inputByte_1)), 
    I_LO := deviceConfig.analogInputLow, 
    I_HI := deviceConfig.analogInputHigh, 
    O_LO := deviceConfig.analogOutputLow, 
    O_HI := deviceConfig.analogOutputHigh
);


// Sensor raw distance
analogInputRaw := (SHL(BYTE_TO_WORD(HwToPlc.inputByte_0),8) OR HwToPlc.inputByte_1);
END_METHOD

METHOD PRIVATE _Scale : REAL
VAR_INPUT
	
	X : REAL;
	I_LO : REAL;
	I_HI : REAL;
	O_LO : REAL;
	O_HI : REAL;
	
END_VAR
IF I_LO = I_HI THEN
	_Scale := O_LO;
ELSE
	_Scale := (O_HI - O_LO) / (I_HI - I_LO) * (LIMIT(I_LO, X, I_HI) - I_LO) + O_LO;
END_IF;
END_METHOD

END_FUNCTION_BLOCK

// ---- Library/Machine/DryEnd/AutomaticOrderChange/FB_AutomaticOrderChange.TcPOU
FUNCTION_BLOCK FB_AutomaticOrderChange
VAR_INPUT
	
	enable						: BOOL;
	executeAOC					: BOOL; 				(*Start automatic order change*)
	executeManualOC				: BOOL;					(*Execute manual order change copy the value from the next order to the current order*)
	rotaryShearCutSensor 		: BOOL;					(*Rotary shear cut sensor*)
	measuringWheelPaperSensor 	: BOOL;					(*Measuring wheel sensor*)
	slitterClearSensor			: BOOL;					(*Slitter clear sensor signal*)
	slitterInPosition			: BOOL;
	rotaryKnifePaperSensor		: BOOL;					(*Rotary knife paper presence sensorl*)
	doubleFacerSpeedMPM			: REAL;	 				(*Line speed in meters per minute (Double facer speed)*)


	configuration					: aocConfig_TypeStruct;		(*Automatic order change configuration parameters*)
	currentOrder					: Order_TypeStruct;				(*Automatic order current order details*)
	nextOrder						: Order_TypeStruct;				(*Automatic order next order details*)

END_VAR
VAR_OUTPUT
	
	error						: BOOL;				(*Error ocurred during automatic order change*)
	aocRunning					: BOOL;				(*Automatic order change running signal*)
	changeOrder					: BOOL;				(*Change order from automatic order change*)
	aocTimeOut					: BOOL;
	
	referenceSwitch				: BOOL;				(*Reference swith between double facer and AOC ramp reference*)
	doubleFacerSpeedUP			: BOOL;				(*Speed up command to double facer*)
	doubleFacerSpeedDown		: BOOL;				(*Speed down command to double facer*)
	doubleFacerStop				: BOOL;				(*Double facer stop command*)
	stopDoubleFacer				: BOOL;				(*Stop command to double facer*)
	rotaryShearCutX1			: BOOL;				(*Rotary shar cut x1 command*)
	slitterChangeOrder			: BOOL;				(*Slitter change order command*)
	flapsChangeOrder			: BOOL;

	lowerLevelStackerDischarge			: BOOL;				(*Top stacker discharge command*)
	upperLevelStackerDischarge			: BOOL;				(*Bottom stacker discharge command*)
	
	rotaryKnifeSpeedRef			: LREAL;
	siltterKnifeSpeedRef		: LREAL;
	siltterScorerSpeedRef		: REAL;

	statusDisplay				: STRING;

END_VAR
VAR
	stateMachine					: WORD;				(*Function block state machine*)
	status							: INT;
	statErrorUserCleared			: BOOL;
	statNotEnabled					: BOOL;
	statFirtsCycle					: BOOL;
	statExecuteManualOC				: BOOL;
	statSpeedDiference				: REAL;				(*Speed diference between double facer and AOC speed*)

	statRotaryKnife1Counter			: DINT;
	statRotaryKnife2Counter			: DINT;


	statPile1Counter				: DINT;
	statPile2Counter				: DINT;


	tempRunningCounter				: DINT;
	statEnableOld					: BOOL;

	instFbCtrlPwm					: FB_CTRL_PWM_OUT_EXT;
	instFbCtrlPwmOutParameters 		: ST_CTRL_PWM_OUT_EXT_PARAMS; (*Configuration of PWM Function block*)

	statePwmInputSignal				: REAL;
	tempDoubleFacerSpeedMPM			: REAL;

	instFbTPRoaryShear						: TP;
	instFbTPSlitter								: TP;
	instFBCtrlRampGenerator					: FB_CTRL_RAMP_GENERATOR;


	statFBCtrlRampGeneratorParams			: ST_CTRL_RAMP_GENERATOR_PARAMS;


	instFbTONSlitterDelay: TON;
	instFbTONStackerDischargeDelay: TON;

	instFbTPStacker1Discharge: TP;
	instFbTPStacker2Discharge: TP;
	tempExecuteAOC: BOOL;
	instFbTONStacker1Discharge: TON;
	instFbTONStacker2Discharge: TON;

	instRotaryShearCutX1TP: TP;
	instChangeSheetLengthTON: TON;
	instAOCTimeOutTON: TON;
	instTONChangeCutLenght: TON;
END_VAR


VAR_IN_OUT



END_VAR

VAR CONSTANT

	STATUS_NO_CALL								: WORD := 16#7000;				(* No call of FB *)
	STATUS_FB_FIRST_CALL						: WORD := 16#7001;				(* First cycle of FB after enabling *)
	STATUS_SUBSEQUENT_CALL						: WORD := 16#7002;				(* FB enabled *)



	STATUS_CHECK_CONDITIONS						: WORD := 16#8000;				(* Check the conditions before start the AOC*)
	STATUS_SAVE_DF_SPEED						: WORD := 16#8001;				(* Saves the current double facer speed and reset variables*)
	STATUS_REDUCE_DF_SPEED						: WORD := 16#8002;				(* Reduce the line speed until the programmed AOC speed*)
	STATUS_ROTARY_SHEAR_CUT_X1					: WORD := 16#8003;				(* Cut the material web*)
	STATUS_INCREASE_DRYEND_SPEED				: WORD := 16#8004;				(* Increase the dryend speed*)
	STATUS_CHANGE_SLT_ORDER						: WORD := 16#8005;				(* FB enabled *)
	STATUS_CHANGE_RK_SHEET_LENGTH				: WORD := 16#8006;				(* FB enabled *)
	STATUS_STK_DISCHARGE						: WORD := 16#8007;				(* FB enabled *)
	STATUS_INCREASE_DF_SPEED					: WORD := 16#8008;				(* FB enabled *)
	STATUS_SYNC_DRYEND_DF_SPEED					: WORD := 16#8009;				(* FB enabled *)
	STATUS_AOC_FINISHED							: WORD := 16#8010;				(* FB enabled *)
	STATUS_AOC_CANCELED							: WORD := 16#8011;				(* FB enabled *)
	STATUS_AOC_ERROR							: WORD := 16#8012;				(* Called if an error occurs during the AOC*)




 END_VAR

(*=================================================================================================
CPNTeck - Automação ind.
(c)Copyright 2022 All Rights Reserved
_______________________________________________________________________________________________________________________________
Library: N/A 
Tested with: C6017 
Engineering: Twincat 3
Restrictions: -
Requirements: N/A
Functionality: This function block offers basic functionalities to control the automatic order change of the machine using
the fallowing functions:
- Reduce the double facer speed
- Execute a single cut in the material web
- Increase the speed of the dryend
- Change the slitter order
- Change the rotary knife sheet lenght
- Execute the stacker discharge of the remaining boards
- Increase the speed of the double facer the the speed that it was before.

Support: fabio@cpnteck.com.br
Note: Parameter comments are only available in language 'English (United States)'
_______________________________________________________________________________________________________________________________
Change log table:
Version  		| Date        			| Expert in charge  			| Changes applied

01.00.01		| 01.02.2026  		| Fabio Campion                	| First released version



==================================================================================================*)

(*------------------------------------------------------------------------------------------------------------------------------------------------------------------------------------*)
(* Enable / disable FB																																			*)
(*------------------------------------------------------------------------------------------------------------------------------------------------------------------------------------*)

(* Reset outputs 																				 *)
(*==========================================================*)
(* Error and valid outputs are reset with falling edge of enable input							 *)

IF NOT enable AND statEnableOld THEN

	(* Reset error and status *)
	error := FALSE;
	status := STATUS_NO_CALL;
	statusDisplay := 'Not running...';

	(* Reset status outputs *)
	error := FALSE;
	aocRunning	 := FALSE;
	//encoderSwitch := FALSE;
	referenceSwitch := FALSE;
	doubleFacerSpeedUP := FALSE;
	doubleFacerSpeedDown := FALSE;
	stopDoubleFacer := FALSE;
	rotaryShearCutX1 := FALSE;
	slitterChangeOrder := FALSE;
	lowerLevelStackerDischarge := FALSE;
	upperLevelStackerDischarge := FALSE;
	instFbTPRoaryShear.IN := FALSE;
	instFbTPSlitter.IN := FALSE;
	instFbTONSlitterDelay.IN := FALSE;
	instFbTONStackerDischargeDelay.IN := FALSE;
	instFbTPStacker1Discharge.IN	:= FALSE;
	instFbTPStacker2Discharge.IN	:= FALSE;
	instFBCtrlRampGenerator.bEnable := FALSE;
	instFBCtrlRampGenerator.fStart := configuration.automaticOrderChangeSpeed;
	instFBCtrlRampGenerator.fTarget := configuration.automaticOrderChangeSpeed;


	rotaryKnifeSpeedRef			:= 0.0;
	siltterKnifeSpeedRef		:= 0.0;

	(* Reset internal variables*)
	statFirtsCycle := FALSE;
	tempRunningCounter := 0;


	statEnableOld := enable;
	RETURN;

(* Check if FB is enabled - first cycle*)
(*===========================================================*)
ELSIF enable AND NOT statEnableOld THEN

	status := STATUS_FB_FIRST_CALL;
	statFirtsCycle := TRUE;
	(* Set old value of enable for edge detection and end execution*)
	statEnableOld := enable;
	RETURN;


(* Check if function block is disabled or UserClearedError is present*)
ELSIF NOT enable THEN

	(*Function block not running*)
	statNotEnabled := TRUE;

ELSE

	(* Function block enabled													    					   *)
	(*===========================================================*)

	(*Function block cycles increment counter*)
	tempRunningCounter := tempRunningCounter + 1;



	(*Execute automatic order change command*)
	IF executeAOC AND NOT tempExecuteAOC THEN

		stateMachine := STATUS_CHECK_CONDITIONS;

	END_IF

	tempExecuteAOC := executeAOC;

	(* Function block state machine											    					   *)
	(*===========================================================*)
	CASE stateMachine OF




	(*----------------------------------------------------------------------------------------------*)
	(* Check the conditions before start the AOC										 *)
	(*----------------------------------------------------------------------------------------------*)
		STATUS_CHECK_CONDITIONS:

		(*Check if there is paper in the machine*)
		IF NOT measuringWheelPaperSensor OR NOT slitterClearSensor OR NOT rotaryKnifePaperSensor THEN

			stateMachine := STATUS_AOC_FINISHED;

		ELSE
			instAOCTimeOutTON.IN := TRUE;
			stateMachine := STATUS_SAVE_DF_SPEED;

		END_IF


	(*----------------------------------------------------------------------------------------------*)
	(* Saves the current running speed of the double facer	to be used latter			 *)
	(*----------------------------------------------------------------------------------------------*)
		STATUS_SAVE_DF_SPEED:

		statusDisplay := 'STATUS_SAVE_DF_SPEED';
		tempDoubleFacerSpeedMPM := doubleFacerSpeedMPM;
		(*instFBCtrlRampGenerator.fTarget := 0;*)
		stateMachine := STATUS_REDUCE_DF_SPEED;


		(*Reset variables*)

		aocRunning := TRUE;
		//encoderSwitch := FALSE;
		doubleFacerSpeedUP := FALSE;
		doubleFacerSpeedDown := FALSE;
		stopDoubleFacer := FALSE;
		
		slitterChangeOrder := FALSE;
		lowerLevelStackerDischarge := FALSE;
		upperLevelStackerDischarge := FALSE;
		instFbTPRoaryShear.IN := FALSE;
		instFbTPSlitter.IN := FALSE;
		instFbTONSlitterDelay.IN := FALSE;
		instFbTONStackerDischargeDelay.IN := FALSE;
		instFbTPStacker1Discharge.IN	:= FALSE;
		instFbTPStacker2Discharge.IN	:= FALSE;

		instFBCtrlRampGenerator.fStart := configuration.automaticOrderChangeSpeed;
		instFBCtrlRampGenerator.fTarget := configuration.automaticOrderChangeSpeed;
		instFBCtrlRampGenerator.bEnable := TRUE;


	(*----------------------------------------------------------------------------------------------*)
	(* Reduce double facer speed to the programmed speed 							 *)
	(*----------------------------------------------------------------------------------------------*)
		STATUS_REDUCE_DF_SPEED:

		statusDisplay := 'STATUS_REDUCE_DF_SPEED';

		IF doubleFacerSpeedMPM > configuration.automaticOrderChangeSpeed THEN

			doubleFacerSpeedDown := instFbCtrlPwm.bPwmOutBitNeg;
			doubleFacerSpeedUP := instFbCtrlPwm.bPwmOutBitPos;

		END_IF

		IF doubleFacerSpeedMPM <= configuration.automaticOrderChangeSpeed THEN

			doubleFacerSpeedDown := FALSE;
			doubleFacerSpeedUP := FALSE;
			stateMachine := STATUS_ROTARY_SHEAR_CUT_X1;

		END_IF

	(*----------------------------------------------------------------------------------------------*)
	(* Cut the web material															 *)
	(*----------------------------------------------------------------------------------------------*)
		STATUS_ROTARY_SHEAR_CUT_X1:

		statusDisplay := 'Cut the material and wait for the sensor of the rotary shear';

		instFbTPRoaryShear.PT := T#1S;
		instFbTPRoaryShear.IN := TRUE;
		
		instRotaryShearCutX1TP.IN := TRUE;



		IF rotaryShearCutSensor THEN
			
			instRotaryShearCutX1TP.IN := FALSE;
			instFbTPRoaryShear.PT := T#1S;
			instFbTPRoaryShear.IN := FALSE;
			referenceSwitch := TRUE;
			stateMachine := STATUS_INCREASE_DRYEND_SPEED;
			changeOrder := TRUE;

		END_IF

		rotaryShearCutX1 := instFbTPRoaryShear.Q;
		instFbTPRoaryShear();

	(*----------------------------------------------------------------------------------------------*)
	(* Increase the dryend speed to clear the slitter and execute the order change	 *)
	(*----------------------------------------------------------------------------------------------*)
	STATUS_INCREASE_DRYEND_SPEED:


		statusDisplay := 'Increase the dryend speed to clear the slitter';

		instFBCtrlRampGenerator.fTarget := configuration.automaticOrderChangeSpeed * configuration.automaticOrderChangeSpeedMult;

		IF NOT measuringWheelPaperSensor THEN

			//encoderSwitch := TRUE;
			stateMachine := STATUS_CHANGE_SLT_ORDER;

		END_IF


	(*----------------------------------------------------------------------------------------------*)
	(* Increase the dryend speed to clear the slitter and execute the order change	 *)
	(*----------------------------------------------------------------------------------------------*)
		STATUS_CHANGE_SLT_ORDER:

		statusDisplay := 'Waiting for the slitter to be clear and change the order (Sensor clear)';

		IF NOT slitterClearSensor THEN

			instFbTPSlitter.PT := T#5S;
			instFbTPSlitter.IN := TRUE;
			stateMachine := STATUS_CHANGE_RK_SHEET_LENGTH;

		END_IF



	(*----------------------------------------------------------------------------------------------*)
	(* Wait until the sensor is clear and change the sheet  length of the rotary knife	 *)
	(*----------------------------------------------------------------------------------------------*)
	STATUS_CHANGE_RK_SHEET_LENGTH:

		statusDisplay := 'Waiting to change rotary knife length (Sensor clear)';

		instTONChangeCutLenght.PT := T#4S;
		instTONChangeCutLenght.IN := TRUE;

		
		instChangeSheetLengthTON.PT := configuration.changeSheetLengthTime;
		instChangeSheetLengthTON.IN := TRUE;
		
		(*Wait until the sensor is clear and change the sheet length*)
		IF NOT rotaryKnifePaperSensor OR instChangeSheetLengthTON.Q THEN
		
		
			flapsChangeOrder := TRUE; (*Adjuste the flaps*)
			instChangeSheetLengthTON.IN := FALSE;
			instChangeSheetLengthTON.IN := FALSE;
			stateMachine := STATUS_STK_DISCHARGE;

		END_IF


	(*----------------------------------------------------------------------------------------------*)
	(* Wait a small delay and discharge the stacker if the ID is diferent				 *)
	(*----------------------------------------------------------------------------------------------*)
	STATUS_STK_DISCHARGE:

	statusDisplay := 'Discharge the stacker if the next order ID is diferent';


		instFbTONStackerDischargeDelay.PT := configuration.stackerDischargeDelay;
		instFbTONStackerDischargeDelay.IN := TRUE;
	
		instFbTONStacker1Discharge.PT := T#2S;
		instFbTONStacker2Discharge.PT := T#2S;
	
		IF instFbTONStackerDischargeDelay.Q THEN
	
			//IF currentOrder.top.id <> nextOrder.top.id THEN

				instFbTONStacker1Discharge.IN := TRUE;
				lowerLevelStackerDischarge := TRUE;
	
			//END_IF
	
	
			//IF currentOrder.bottom.id <> nextOrder.bottom.id THEN
	
				instFbTONStacker2Discharge.IN := TRUE;
				upperLevelStackerDischarge := TRUE;

			//END_IF
	
		END_IF

		IF instFbTONStackerDischargeDelay.Q  THEN

			IF  instFbTONStacker1Discharge.Q OR instFbTONStacker2Discharge.Q THEN

				lowerLevelStackerDischarge := FALSE;
				upperLevelStackerDischarge := FALSE;
				instFbTONStackerDischargeDelay.IN := FALSE;
				instFbTONStacker1Discharge.IN := FALSE;
				instFbTONStacker2Discharge.IN := FALSE;
				currentOrder := nextOrder;
				stateMachine := STATUS_AOC_FINISHED;

			END_IF
	
		END_IF



	instFbTONStacker1Discharge();
	instFbTONStacker2Discharge();
	instFbTONStackerDischargeDelay();




	(*----------------------------------------------------------------------------------------------*)
	(* AOC Finished																	 *)
	(*----------------------------------------------------------------------------------------------*)
	STATUS_AOC_FINISHED:

	statusDisplay := 'STATUS_AOC_FINISHED...';
	
	aocRunning	 := FALSE;
	//encoderSwitch := FALSE;
	referenceSwitch := FALSE;
	doubleFacerSpeedUP := FALSE;
	doubleFacerSpeedDown := FALSE;
	stopDoubleFacer := FALSE;
	instRotaryShearCutX1TP.IN := FALSE;
	slitterChangeOrder := FALSE;
	flapsChangeOrder := FALSE; (*Adjuste the flaps*)

	lowerLevelStackerDischarge := FALSE;
	upperLevelStackerDischarge := FALSE;
	instFbTPRoaryShear.IN := FALSE;
	instFbTPSlitter.IN := FALSE;
	instFbTPSlitter.IN := FALSE;
	instFbTONSlitterDelay.IN := FALSE;
	instFbTONStackerDischargeDelay.IN := FALSE;
	instFbTPStacker1Discharge.IN	:= FALSE;
	instFbTPStacker2Discharge.IN	:= FALSE;
	instFBCtrlRampGenerator.bEnable := FALSE;
	instFBCtrlRampGenerator.fTarget := configuration.automaticOrderChangeSpeed;
	changeOrder := FALSE;
	instAOCTimeOutTON.IN := FALSE;


	END_CASE

END_IF



	(*----------------------------------------------------------------------------------------------*)
	(* PWM FunctionBlock call															 *)
	(*----------------------------------------------------------------------------------------------*)

	(*Parameters configuration*)
	instFbCtrlPwmOutParameters.tTaskCycleTime := configuration.taskCycleTime;
	instFbCtrlPwmOutParameters.tMinOnTime := T#100MS;
	instFbCtrlPwmOutParameters.tMinOffTime := T#100MS;
	instFbCtrlPwmOutParameters.tPWMPeriod := T#1S;

	(*Speed error calculation for the PWM input*)
	statSpeedDiference := configuration.automaticOrderChangeSpeed - doubleFacerSpeedMPM;

	(*Pwm input calculation and LIMIT*)
	statePwmInputSignal := LIMIT (-100 , (statSpeedDiference * configuration.speedErrorGain ), 100);

	(*PWM Function block call*)
	instFbCtrlPwm(
		fPwmInput := -20,
		eMode:= eCTRL_MODE_ACTIVE,
		stParams:= instFbCtrlPwmOutParameters );


	(*----------------------------------------------------------------------------------------------*)
	(* Ramp FunctionBlock call															 *)
	(*----------------------------------------------------------------------------------------------*)
	(*Function block output call*)

		statFBCtrlRampGeneratorParams.fVeloPos := configuration.rampUpTimeSec;
		statFBCtrlRampGeneratorParams.fVeloNeg := configuration.rampDownTimeSec;
		statFBCtrlRampGeneratorParams.tCtrlCycleTime := configuration.controlerCycleTime;
		statFBCtrlRampGeneratorParams.tTaskCycleTime := configuration.taskCycleTime;

		instFBCtrlRampGenerator(
			stParams:= statFBCtrlRampGeneratorParams);


		rotaryKnifeSpeedRef := instFBCtrlRampGenerator.fOut * configuration.rotaryKnifeSpeedMult;
		siltterKnifeSpeedRef	 := instFBCtrlRampGenerator.fOut	* configuration.slitterSpeedMult;
	


	(*----------------------------------------------------------------------------------------------*)
	(* Execute manual order change																	 *)
	(*----------------------------------------------------------------------------------------------*)

	IF executeManualOC AND NOT statExecuteManualOC THEN

		currentOrder := nextOrder;

	END_IF

	statExecuteManualOC := executeManualOC;

	
	instRotaryShearCutX1TP(PT:=T#500MS,Q=>rotaryShearCutX1);
	instFbTPSlitter(Q=>slitterChangeOrder);
	
	instChangeSheetLengthTON();
	
	(*----------------------------------------------------------------------------------------------*)
	(* AOC Timeout																	 *)
	(*----------------------------------------------------------------------------------------------*)
	
	IF instAOCTimeOutTON.Q THEN
		
		instAOCTimeOutTON.IN := FALSE;
		stateMachine := STATUS_AOC_FINISHED;
		aocTimeOut := TRUE;

	
	END_IF
	
	instAOCTimeOutTON(PT:=configuration.aocTimeout);

END_FUNCTION_BLOCK

// ---- Library/Machine/DryEnd/AutomaticOrderChange/FB_AutomaticOrderChange_V1_BAK.TcPOU
FUNCTION_BLOCK FB_AutomaticOrderChange_V1_BAK
VAR_INPUT
    // ==============================
    // CONTROL
    // ==============================
    enable                      : BOOL;
    executeAOC                  : BOOL;     // Start automatic order change (level trigger)

    // ==============================
    // SENSORS
    // ==============================
    rotaryShearCutSensor        : BOOL;     // Rotary shear cut sensor
    measuringWheelPaperSensor   : BOOL;     // Measuring wheel sensor
    slitterPaperPresenceSensor  : BOOL;     // Slitter paper presence
    rotaryKnifePaperSensor      : BOOL;     // Rotary knife paper presence

    // ==============================
    // PROCESS VALUES
    // ==============================
    lineSpeedMPM                : REAL;     // Line speed [m/min]
    configuration               : aocConfig_TypeStruct; // AOC configuration parameters
END_VAR

VAR_IN_OUT
    currentOrder                : Order_TypeStruct;     // Current order details
    nextOrder                   : Order_TypeStruct;     // Next order details
END_VAR

VAR_OUTPUT
    // ==============================
    // STATUS
    // ==============================
    error                       : BOOL;
    aocRunning                  : BOOL;
    aocTimeOut                  : BOOL;
    statusDisplay               : STRING;

	
	rotaryShearCutX1Timeout		: BOOL;
	measuringWheelClearTimeout	: BOOL;
	slitterClearTimeout			: BOOL;
	rotaryKnifeClarTimeout		: BOOL;
	
    // ==============================
    // MACHINE COMMANDS
    // ==============================
    referenceSwitch             : BOOL;     // Switch between double facer and AOC ramp reference
    doubleFacerSpeedUP          : BOOL;
    doubleFacerSpeedDown        : BOOL;

    // ==============================
    // TRIGGERS / PULSES
    // ==============================
    rotaryShearCutX1            : BOOL;
    executePositioning          : BOOL;
    topStackerDischarge         : BOOL;
    bottomStackerDischarge      : BOOL;

    // ==============================
    // SPEED REFERENCES
    // ==============================
    rotaryKnifeSpeedRef         : LREAL;
    slitterKnifeSpeedRef        : LREAL;
    slitterScorerSpeedRef       : REAL;
END_VAR

VAR
    // ==============================
    // STATE MACHINE
    // ==============================
    stateMachine                : WORD;

    // ==============================
    // EDGE / INTERNAL LATCHES
    // ==============================
    enableOld                   : BOOL;
    executeAOC_Old              : BOOL;
    rExecuteAOC                 : BOOL;      // rising edge of executeAOC

    // ==============================
    // REQUESTS (drive FB inputs)
    // ==============================
    reqTpRotaryShear            : BOOL;
    reqTpExecutePositioning     : BOOL;
    reqTpStackerTop             : BOOL;
    reqTpStackerBottom          : BOOL;

    reqTonSlitterDelay          : BOOL;
    reqTonStackerDelay          : BOOL;
    reqTonChangeSheetLength     : BOOL;

    // ==============================
    // FUNCTION BLOCK INSTANCES
    // ==============================
    tpRotaryShear               : TP;
    tpExecutePositioning        : TP;
    tpStackerTop                : TP;
    tpStackerBottom             : TP;

    tonSlitterPresenceDelay     : TON;
    tonStackerDischargeDelay    : TON;
    tonChangeSheetLength        : TON;

    tonAocTimeout               : TON;

    instFB_Gen_SRamp            : FB_Gen_SRamp;
    instGEN_PULSESpeedCtrl      : GEN_PULSE;

    lineSpeedMPMRamp            : REAL;

